TYPE ST145_Cylinders_e : ST110_Cylinders_e;
END_TYPE

(* stored: Version 1.1.0.1, ProductVersion 3.1.4024.6
   EnumerationTextList ST145_Cylinders_e: Id {70c2502a-ef8a-435a-b832-de209e1efda3} *)
